{attribute 'qualified_only'}
VAR_GLOBAL
	MachineIsActive: BOOL;
	MachineIsRunning : BOOL;
	Emergency: BOOL;
	PBStart : BOOL;
	PBStop : BOOL;
	PBEmergency: BOOL;
END_VAR

(* stored: Version 1.1.0.1, ProductVersion 3.1.4024.12
   GVL GVL: Id {48064612-5b8f-4724-8ff4-d96204304ecb} *)
